{attribute 'GeneratedUsingTerminal: BK1250-0000-0000'}
{attribute addProperty BoxType "BK1250-0000-0000"}
{attribute addProperty Id "CouplerCtrlAT %I*UINT0"}
{attribute addProperty CRC "3636114355"}
{attribute addProperty Size "0"}
TYPE Outputs_D8BAB3B3 EXTENDS InputBase_8311D824 :
STRUCT
	{attribute addProperty Name "CouplerCtrl"}
	CouplerCtrl AT %I* : UINT;
END_STRUCT
END_TYPE

(* stored: Version 1.2.0.0, ProductVersion 3.1.4024.9
   DUT Outputs_D8BAB3B3: Id {9e73058e-2022-41dd-bbb3-32681bd074d3} *)
